{attribute addProperty BoxType "EP2816-0008-0019"}
{attribute addProperty Id "DIG_Diag_Inputs_ChannelAT %I*ARRAY[0..1] OF DIG_Diag_Inputs_Channel_AC4A9AF0128160DIG_Inputs_DeviceAT %I*DIG_Inputs_Device_30BACB404050DIG_Outputs_ChannelAT %Q*ARRAY[0..1] OF DIG_Outputs_Channel_33B76376128160DIG_Outputs_DeviceAT %Q*DIG_Outputs_Device_735003021620WcStateAT %I*WcState_F855686C1620InfoDataAT %I*InfoData_BC63D37F80100"}
{attribute addProperty CRC "2364611730"}
{attribute addProperty SizeInBites "408"}
{attribute addProperty SizeInBytes "51"}
TYPE EP2816_1A393DE7 :
STRUCT
	{attribute addProperty Name "DIG_Diag_Inputs_Channel"}
	DIG_Diag_Inputs_Channel : ARRAY[0..1] OF DIG_Diag_Inputs_Channel_AC4A9AF0;
	{attribute addProperty Name "DIG_Inputs_Device"}
	DIG_Inputs_Device : DIG_Inputs_Device_30BACB40;
	{attribute addProperty Name "DIG_Outputs_Channel"}
	DIG_Outputs_Channel : ARRAY[0..1] OF DIG_Outputs_Channel_33B76376;
	{attribute addProperty Name "DIG_Outputs_Device"}
	DIG_Outputs_Device : DIG_Outputs_Device_73500302;
	{attribute addProperty Name "WcState"}
	WcState : WcState_F855686C;
	{attribute addProperty Name "InfoData"}
	InfoData : InfoData_BC63D37F;
END_STRUCT
END_TYPE

(* stored: Version 1.2.0.0, ProductVersion 3.1.4024.9
   DUT EP2816_1A393DE7: Id {83a82e74-068c-4908-8ed6-340fcabb8f23} *)
